{attribute addProperty BoxType "EJ2521-0224-0016"}
{attribute addProperty Id "ControlAT %Q*Control_E8AFF3DF1620Set_counter_valueAT %Q*UINT16217"}
{attribute addProperty CRC "1552329373"}
{attribute addProperty SizeInBites "32"}
{attribute addProperty SizeInBytes "4"}
TYPE ENC_Control_compact_5C86AA9D :
STRUCT
	{attribute addProperty Name "Control"}
	Control AT %Q* : Control_E8AFF3DF;
	{attribute addProperty Name "Set_counter_value"}
	Set_counter_value AT %Q* : UINT;
END_STRUCT
END_TYPE

(* stored: Version 1.2.0.0, ProductVersion 3.1.4024.9
   DUT ENC_Control_compact_5C86AA9D: Id {0c3e6a09-98b6-4ac2-b0b6-4132e55566cb} *)
